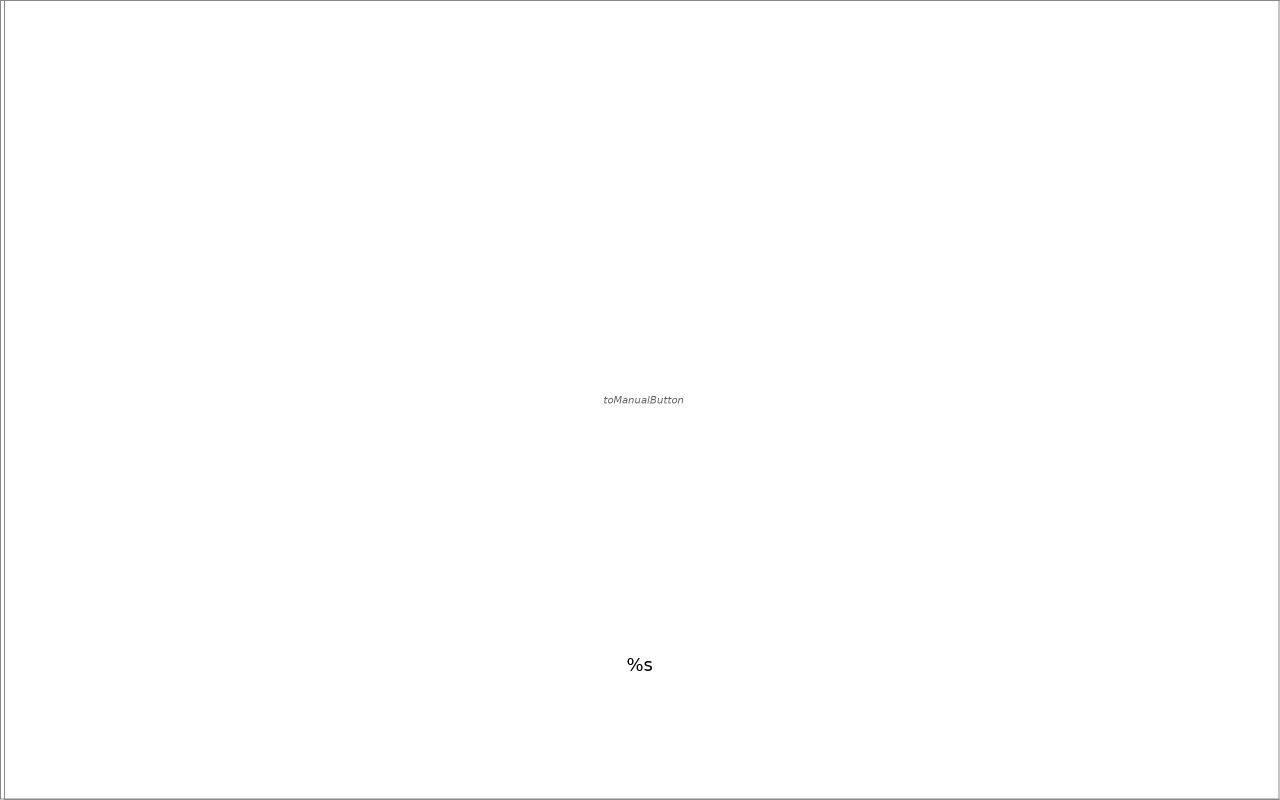
VISUALIZATION LogoScreenBlanc_SVG  // 1280x800
    Frame (4,0 1280x800)
        shows toManualButton()
    Textfield (240,650 800x30), "%s", tooltip "Operator messagages", text variable: GVL_Message.sOPeratorMessage
END_VISUALIZATION

(* stored: Version 1.1.0.1, ProductVersion 3.1.4024.10
   Visu LogoScreenBlanc_SVG: Id {fe6a7024-be80-43a8-beb7-86e60a2e1e58} *)
